// TIA Portal V19 export
TYPE "TAx_Pos_Ctrl"
// stored: Access Published
   STRUCT
      SafeStop : Bool;   // 1 / Emergency stop (device in safe state)
      Rst : Bool;   // Reset alarms
      RstHW : Bool;   // Reset hardware
      Power : Bool;   // Power axis command
      Homing : Bool;
      VelocityPositionControlled : Bool;
      MovePlus : Bool;
      MoveMinus : Bool;
      MoveAbsolute : Bool;
      ExtControl : Bool;   // Axis is controlled from external istruction (MC_Halt not work)
      HomeMode : Int;   // see MC Home
      HomePosition : LReal;
      Velocity : LReal;
      Acceleration : LReal;
      Deceleration : LReal;
      Jerk : LReal;
      MoveAbsTarget : LReal;
      MoveAbsDirection : Int := 3;
   END_STRUCT;
END_TYPE
